FUNCTION_BLOCK GoToManual IMPLEMENTS I_Transitive
VAR
    _currentState : POINTER TO I_SD_ValveState;
    _nextState : REFERENCE TO ManualState;
END_VAR

METHOD FB_init : BOOL
VAR_INPUT
	bInitRetains : BOOL; // if TRUE, the retain variables are initialized (warm start / cold start)
	bInCopyCode : BOOL;  // if TRUE, the instance afterwards gets moved into the copy code (online change)
    currentState : POINTER TO I_SD_ValveState;
    nextState : REFERENCE TO ManualState;
END_VAR
_currentState := currentState;
_nextState REF= nextState;
END_METHOD

METHOD Transit
_currentState^ := _nextState;
END_METHOD

END_FUNCTION_BLOCK

(* stored: Version 1.1.0.1, ProductVersion 3.1.4024.12
   POU GoToManual: Id {a34a26cd-043e-4215-9a1e-4ad186729859}, SpecialFunc None
   Method FB_init: Id {de399ccd-7055-4c9a-a9a3-844210412fae}
   Method Transit: Id {1d5488a2-b1ed-4e73-9743-cf72b31206a5} *)
